// X9 must stay quiet here, and this is why the pin matchers are anchored. Every name
// below ends in Enable or Done but names the completion of one specific operation
// rather than a PLCopen command pin. A substring match fires on all of them: measured
// on one real project, loosening the matcher added 13 findings, every one of them wrong.
FUNCTION_BLOCK FB_NamedCompletions
VAR_INPUT
    ibSimulationEnabled : BOOL;     // a mode flag, not the PLCopen Enable family
    CFG_bEnableActivateRemoteButton : BOOL;
END_VAR
VAR_OUTPUT
    obHomingDone : BOOL;            // this axis finished homing; says nothing about the FB
    obInfo_CalibrationDone : BOOL;
END_VAR

obHomingDone := ibSimulationEnabled;
obInfo_CalibrationDone := CFG_bEnableActivateRemoteButton AND obHomingDone;

END_FUNCTION_BLOCK

(* stored: Version 1.1.0.1, ProductVersion 3.1.4024.0
   POU FB_NamedCompletions: Id {3e9a1b40-77c2-4f16-9a03-1d5b8c2e4475}, SpecialFunc None *)
